{attribute 'GeneratedUsingTerminal: EL6201-0000-0017'}
{attribute addProperty BoxType "EL6201-0000-0017"}
{attribute addProperty Id "Slave_1_InputsAT %I*Slave_1_Inputs_2C3058A88Slave_2_InputsAT %I*Slave_2_Inputs_413F454C8Slave_3_InputsAT %I*Slave_3_Inputs_9985457D8Slave_4_InputsAT %I*Slave_4_Inputs_9B217E848Slave_5_InputsAT %I*Slave_5_Inputs_439B7EB58Slave_6_InputsAT %I*Slave_6_Inputs_2E9463518Slave_7_InputsAT %I*Slave_7_Inputs_F62E63608Slave_8_InputsAT %I*Slave_8_Inputs_2BDC14A38Slave_9_InputsAT %I*Slave_9_Inputs_F36614928Slave_10_InputsAT %I*Slave_10_Inputs_01E65E7D8Slave_11_InputsAT %I*Slave_11_Inputs_D274DB978Slave_12_InputsAT %I*Slave_12_Inputs_A202481E8Slave_13_InputsAT %I*Slave_13_Inputs_7190CDF48Slave_14_InputsAT %I*Slave_14_Inputs_42EF6F0C8Slave_15_InputsAT %I*Slave_15_Inputs_917DEAE68Slave_16_InputsAT %I*Slave_16_Inputs_E10B796F8Slave_17_InputsAT %I*Slave_17_Inputs_3299FC858Slave_18_InputsAT %I*Slave_18_Inputs_87F43C9F8Slave_19_InputsAT %I*Slave_19_Inputs_5466B9758Slave_20_InputsAT %I*Slave_20_Inputs_97C1CA9A8Slave_21_InputsAT %I*Slave_21_Inputs_44534F708Slave_22_InputsAT %I*Slave_22_Inputs_3425DCF98Slave_23_InputsAT %I*Slave_23_Inputs_E7B759138Slave_24_InputsAT %I*Slave_24_Inputs_D4C8FBEB8Slave_25_InputsAT %I*Slave_25_Inputs_075A7E018Slave_26_InputsAT %I*Slave_26_Inputs_772CED888Slave_27_InputsAT %I*Slave_27_Inputs_A4BE68628Slave_28_InputsAT %I*Slave_28_Inputs_11D3A8788Slave_29_InputsAT %I*Slave_29_Inputs_C2412D928Slave_30_InputsAT %I*Slave_30_Inputs_199C4DAA8Slave_31_InputsAT %I*Slave_31_Inputs_CA0EC8408"}
{attribute addProperty CRC "2133338277"}
{attribute addProperty Size "248"}
TYPE ASI_Inputs_Device_7F2828A5 EXTENDS InputBase_8311D824 :
STRUCT
	{attribute addProperty Name "Slave_1_Inputs"}
	Slave_1_Inputs AT %I* : Slave_1_Inputs_2C3058A8;
	{attribute addProperty Name "Slave_2_Inputs"}
	Slave_2_Inputs AT %I* : Slave_2_Inputs_413F454C;
	{attribute addProperty Name "Slave_3_Inputs"}
	Slave_3_Inputs AT %I* : Slave_3_Inputs_9985457D;
	{attribute addProperty Name "Slave_4_Inputs"}
	Slave_4_Inputs AT %I* : Slave_4_Inputs_9B217E84;
	{attribute addProperty Name "Slave_5_Inputs"}
	Slave_5_Inputs AT %I* : Slave_5_Inputs_439B7EB5;
	{attribute addProperty Name "Slave_6_Inputs"}
	Slave_6_Inputs AT %I* : Slave_6_Inputs_2E946351;
	{attribute addProperty Name "Slave_7_Inputs"}
	Slave_7_Inputs AT %I* : Slave_7_Inputs_F62E6360;
	{attribute addProperty Name "Slave_8_Inputs"}
	Slave_8_Inputs AT %I* : Slave_8_Inputs_2BDC14A3;
	{attribute addProperty Name "Slave_9_Inputs"}
	Slave_9_Inputs AT %I* : Slave_9_Inputs_F3661492;
	{attribute addProperty Name "Slave_10_Inputs"}
	Slave_10_Inputs AT %I* : Slave_10_Inputs_01E65E7D;
	{attribute addProperty Name "Slave_11_Inputs"}
	Slave_11_Inputs AT %I* : Slave_11_Inputs_D274DB97;
	{attribute addProperty Name "Slave_12_Inputs"}
	Slave_12_Inputs AT %I* : Slave_12_Inputs_A202481E;
	{attribute addProperty Name "Slave_13_Inputs"}
	Slave_13_Inputs AT %I* : Slave_13_Inputs_7190CDF4;
	{attribute addProperty Name "Slave_14_Inputs"}
	Slave_14_Inputs AT %I* : Slave_14_Inputs_42EF6F0C;
	{attribute addProperty Name "Slave_15_Inputs"}
	Slave_15_Inputs AT %I* : Slave_15_Inputs_917DEAE6;
	{attribute addProperty Name "Slave_16_Inputs"}
	Slave_16_Inputs AT %I* : Slave_16_Inputs_E10B796F;
	{attribute addProperty Name "Slave_17_Inputs"}
	Slave_17_Inputs AT %I* : Slave_17_Inputs_3299FC85;
	{attribute addProperty Name "Slave_18_Inputs"}
	Slave_18_Inputs AT %I* : Slave_18_Inputs_87F43C9F;
	{attribute addProperty Name "Slave_19_Inputs"}
	Slave_19_Inputs AT %I* : Slave_19_Inputs_5466B975;
	{attribute addProperty Name "Slave_20_Inputs"}
	Slave_20_Inputs AT %I* : Slave_20_Inputs_97C1CA9A;
	{attribute addProperty Name "Slave_21_Inputs"}
	Slave_21_Inputs AT %I* : Slave_21_Inputs_44534F70;
	{attribute addProperty Name "Slave_22_Inputs"}
	Slave_22_Inputs AT %I* : Slave_22_Inputs_3425DCF9;
	{attribute addProperty Name "Slave_23_Inputs"}
	Slave_23_Inputs AT %I* : Slave_23_Inputs_E7B75913;
	{attribute addProperty Name "Slave_24_Inputs"}
	Slave_24_Inputs AT %I* : Slave_24_Inputs_D4C8FBEB;
	{attribute addProperty Name "Slave_25_Inputs"}
	Slave_25_Inputs AT %I* : Slave_25_Inputs_075A7E01;
	{attribute addProperty Name "Slave_26_Inputs"}
	Slave_26_Inputs AT %I* : Slave_26_Inputs_772CED88;
	{attribute addProperty Name "Slave_27_Inputs"}
	Slave_27_Inputs AT %I* : Slave_27_Inputs_A4BE6862;
	{attribute addProperty Name "Slave_28_Inputs"}
	Slave_28_Inputs AT %I* : Slave_28_Inputs_11D3A878;
	{attribute addProperty Name "Slave_29_Inputs"}
	Slave_29_Inputs AT %I* : Slave_29_Inputs_C2412D92;
	{attribute addProperty Name "Slave_30_Inputs"}
	Slave_30_Inputs AT %I* : Slave_30_Inputs_199C4DAA;
	{attribute addProperty Name "Slave_31_Inputs"}
	Slave_31_Inputs AT %I* : Slave_31_Inputs_CA0EC840;
END_STRUCT
END_TYPE

(* stored: Version 1.2.0.0, ProductVersion 3.1.4024.9
   DUT ASI_Inputs_Device_7F2828A5: Id {d7972cf8-7dbd-4458-8cfa-d98ecf519c81} *)
